{attribute 'qualified_only'}
{attribute 'strict'}
TYPE BufferState :
(
	INIT, IDLE, STORING, FULL
);
END_TYPE

(* stored: Version 1.1.0.1, ProductVersion 3.1.4024.12
   DUT BufferState: Id {f9e34e67-7bcf-4e6d-b22e-cf8363f12bc8} *)
